Staubli VAL3: advance.pjx

--- advance.pjx ---
Parameters version=s7.2.1 stackSize=5000 millimeterUnit=true
Program file=findLastPathPos.pgx
Program file=language.pgx
Program file=loadPage.pgx
Program file=main.pgx
Program file=onEnterEvent.pgx
Program file=onExit.pgx
Program file=onF1Event.pgx
Program file=onF2Event.pgx
Program file=onF3Event.pgx
Program file=onF4Event.pgx
Program file=onF5Event.pgx
Program file=onF6Event.pgx
Program file=onF7Event.pgx
Program file=onF8Event.pgx
Program file=onStart.pgx
Program file=passwd.pgx
Program file=refresh.pgx
Program file=refreshDynamic.pgx
Program file=refreshExport.pgx
Program file=refreshImport.pgx
Program file=refreshStatic.pgx
Program file=settings.pgx
Data file=advance.dtx
Library alias=use path=Disk://kernel/userPage/userPage.pjx
Library alias=use2 path=Disk://kernel/userpage/userpage.pjx
Library alias=language path=Disk://kernel/language/language.pjx
Library alias=saveData path=Disk://saveData/saveData.pjx
Library alias=out path=Disk://instruction/inputOutput/OUT/OUT.pjx
Library alias=cycleStatus path=Disk://cycleStatus/cycleStatus.pjx
Library alias=tcp path=Disk://kernel/tool/tool.pjx
Library alias=page path=Disk://kernel/template/page/page.pjx
Type name=FrameItem path=Disk://kernel/template/FrameItem/FrameItem.pjx

--- advance.dtx ---
num nIndex
num nIndexExport
num nIndexImport
num nIndexPreset
num nKey
public num nPage
num nRefresh
num nTime = 1
num nView
num nViewExport
num nViewImport
string sEventExport
string sEventImport
string sExport
string sImport
public string sItems
string sMenu
string sMessage
string sMenu8[8]
bool bButton[8]
frame fFrame = {fatherId=world[0]}

--- main.pgx ---
public program main()
  local bool l_bSave
begin
  // INIT
  call onStart()
  // LOOP UNTIL nKey=255
  do
    call refresh()
    nKey=getKey()
    switch nKey
      case 271
        // GUN SELECTION
        call onF1Event(l_bSave)
      break
      case 272
        // LANGUAGE
        call onF2Event(l_bSave)
      break
      case 273
        //
        call onF3Event()
      break
      case 274
        //
        call onF4Event()
      break
      case 275
        //
        call onF5Event()
      break
      case 276
        // PLC
        call onF6Event(l_bSave)
      break
      case 277
        // PROFIILE
        call onF7Event(l_bSave)
      break
      case 278
        //
        call onF8Event()
      break
      case 270
        // NOTHING
        call onEnterEvent()
      break
    endSwitch
    //release the resource
    delay(0)
  until nKey==255
  // on Exit
  call onExit(l_bSave)
end

--- findLastPathPos.pgx ---
program findLastPathPos(string x_sPath (dimensions=1), num& x_nPos[] (dimensions=1))
  local num l_nPos[2]
  local string l_sPath
begin
  // get the trajType
  l_sPath=x_sPath
  x_nPos=0
  do
    l_nPos=find(l_sPath,"/")
    if l_nPos==-1
      l_nPos=find(l_sPath,"\")
    endIf
    if l_nPos!=-1
      x_nPos=x_nPos+l_nPos+1
      l_nPos[1]=l_nPos
      l_sPath=right(l_sPath,len(l_sPath)-l_nPos-1)
    endIf
  until l_nPos==-1
  // came back one
  x_nPos=x_nPos-l_nPos[1]-1
end

--- language.pgx ---
program language()
  local num l_nIndex
  local string l_sEvent
  local num i
  local string l_sMessage
begin
  //
  //  Select and change the language
  //
  call use:clear(0,13)
  call use:setView(false)
  // scan it
  libList(language:libPath(),sMessage)
  // clean
  for i=0 to size(sMessage)-1
    if find(sMessage[i],".")!=-1
      delete(sMessage[i])
      i=i-1
    endIf
  endFor
  call language:message(l_sMessage,50)
  call use:setSizeList(19,0,19,11)
  call use:listcreate(l_sMessage)
  // show it
  for i=0 to (size(sMessage)-1)
    l_sEvent=sMessage[i]
    call use:listadd(l_sEvent)
    if saveData:language==sMessage[i]
      l_nIndex=i
    endIf
  endFor
  // update the list
  use:nView=l_nIndex
  call use:listupdate(0)
  // scan for a button
  do
    i=get()
    call use:listevent(i,l_nIndex,l_sEvent)
  until i==270 or i==255
  if (i==270) and l_nIndex!=-1
    saveData:language=l_sEvent
    logMsg("[KERNEL] INTERFACE:Change language to "+l_sEvent)
    // set the language
    call language:setLanguage(language:libPath()+"/"+saveData:language)
  else
    call use:nullKey(i)
  endIf
end

--- loadPage.pgx ---
program loadPage(string x_sPage, string& x_sItems[])
// load the next page
  local num i
  local string l_sMessage
begin
  // look if the page libload is correct
  i=page:libLoad(x_sPage)
  delay(0)
  if i!=0
    logMsg("[KERNEL] INTERFACE:PAGE LIBLOAD "+x_sPage+" result "+toString("",i))
    call language:message(l_sMessage,-7)
    popUpMsg(l_sMessage+x_sPage+" ; "+toString("",i))
  else
    // copy all the field from x_sItems to the next page
    call use:stringCopy(x_sItems,page:sItems)
    call page:main()
  endIf
end

--- onEnterEvent.pgx ---
program onEnterEvent()
begin
  //
end

--- onExit.pgx ---
program onExit(bool x_bSave (dimensions=1))
  local num i
begin
  // save the saveData module
  if x_bSave
    if saveData:libSave()!=0
      delay(0.5)
      i=saveData:libSave()
      if i!=0
        popUpMsg("libsave saveData error: "+toString("",i))
        logMsg("[KERNEL] ADVANCE:Error saving saveData "+toString("",i))
      endIf
    endIf
  endIf
  //
  call use:nullKey(nKey)
end

--- onF1Event.pgx ---
program onF1Event(bool& x_bSave[])
  local string l_sParameter
  local string l_sItem
  local num l_nKey
  local num l_nIndex
  local string l_sPage
  local string l_sEvent
  local num i
begin
  // look if the bButton is enable
  if bButton[0]
    //
    // TOOL / FRAME SELECTION
    //
    call use:setSizeList(0,9,10,2)
    call use:listcreate("")
    // TOOL
    call language:message(l_sItem,124)
    call use:listadd(l_sItem)
    l_sItem="FRAME"
    call use:listadd(l_sItem)
    call use:listupdate(0)
    // get the key
    do
      l_nKey=get()
      call use:listevent(l_nKey,l_nIndex,l_sEvent)
    until l_nKey==270 or l_nKey==255
    // check the Enter key pressure
    if l_nKey==270
      switch l_nIndex
        case 0
          // Select the tool
          l_sPage="Disk://kernel/page/tool"
          call loadPage(l_sPage,l_sItem)
        break
        case 1
          // Select the Frame
          l_sPage="Disk://kernel/page/frame"
          call loadPage(l_sPage,l_sItem)
        break
      endSwitch
    endIf
    logMsg("[KERNEL] INTERFACE:PAGE Advance")
    x_bSave=true
  endIf
end

--- onF2Event.pgx ---
program onF2Event(bool& x_bSave[] (dimensions=1))
begin
  // look if the bButton is enable
  if bButton[1]
    //
    // CHANGE THE settings
    //
    setTextMode(1)
    call use:type(0,4,"F2 "+sMenu[1])
    setTextMode(0)
    call settings()
    use:bUseRefresh=true
    x_bSave=true
  endIf
end

--- onF3Event.pgx ---
program onF3Event()
  local string l_sMessage[2]
  local bool l_bImport
  local string l_sPath[2]
  local num l_nKey
  local bool l_bDone
  local num l_nOldValue[4]
  local num i
  local string l_sButton[2]
  local string l_sItem
  local string l_sType
begin
  //
  // look if the bButton is enable
  if bButton[2]
    if libList("USB0://",sImport)
      l_bImport=false
      //
      //  importing file
      //
      // get the path
      l_sPath="Disk://../usrapp/"
      //
      l_sPath[1]="USB0://"
      //
      title("< RESTORE / BACKUP >")
      cls()
      // copy the value
      l_nOldValue[2]=nIndexImport
      l_nOldValue[3]=nViewImport
      l_nOldValue=nIndex=0
      l_nOldValue[1]=nView
      //
      // IMPORT
      call use2:setSizeList(0,0,17,11)
      call use2:listcreate("USB")
      // paste the value
      nIndexImport=l_nOldValue[2]
      nViewImport=l_nOldValue[3]
      call refreshImport(false,l_sPath)
      // EXPORT
      call use:setSizeList(19,0,19,11)
      call use:listcreate("ROBOT")
      // paste the value
      nIndex=l_nOldValue=0
      nView=l_nOldValue[1]
      call refreshExport(true,l_sPath)
      l_sType="<<<<"
      call use:type(17,12,l_sType)
      //
      do
        call use:clear(0,13)
        call use:typeMenu(8,"COPY")
        l_nKey=get()
        switch l_nKey
          case 264
            l_bImport=true
            //refresh
            call refreshExport(false,l_sPath)
            call refreshImport(true,l_sPath)
            l_sType=">>>>"
            call use:type(17,12,l_sType)
          break
          case 268
            l_bImport=false
            //refresh
            //call refreshExport(true,l_sPath)
            call refreshImport(false,l_sPath)
            call refreshExport(true,l_sPath)
            l_sType="<<<<"
            call use:type(17,12,l_sType)
          break
        endSwitch
        // swich from import to export
        if l_bImport
          //
          // IMPORT
          //
          call use2:listevent(l_nKey,nIndexImport,sEventImport)
          nViewImport=use2:nView
          //
          if l_nKey>=259 and l_nKey<=278
            if l_nKey==278
              // look for already exist
              l_bDone=true
              for i=0 to size(sExport)-1
                if sExport[i]==sEventImport
                  call language:message(l_sMessage,11)
                  // get the yes_no button Key
                  call language:getYesNo(l_sButton)
                  // ask the question
                  call use:yes_no(l_sMessage+"#"+l_sPath+sEventImport,l_sButton,l_bDone)
                  i=size(sExport)-1
                endIf
              endFor
              //
              if l_bDone
                call language:message(l_sMessage,10)
                // show that will take several minute
                if find(sEventExport,"usrapp")!=-1
                  call language:message(l_sMessage[1],-9)
                  l_sMessage=l_sMessage+"#"+l_sMessage[1]
                endIf
                call use:timerDialog(l_sMessage+"#"+l_sPath+sEventImport,0)
                l_bDone=$copy(l_sPath[1]+sEventImport,l_sPath+sEventImport)
                if !l_bDone
                  call language:message(l_sMessage,-6)
                  call use:timerDialog(l_sMessage+"#"+l_sPath+sEventImport,2)
                endIf
              endIf
              // refresh backward
              cls()
              call refreshExport(false,l_sPath)
              call refreshImport(true,l_sPath)
              l_sType=">>>>"
              call use:type(17,12,l_sType)
            endIf
          endIf
          //
        else
          //
          //  EXPORT
          //
          call use:listevent(l_nKey,nIndex,sEventExport)
          nView=use:nView
          //
          if l_nKey>=259 and l_nKey<=278
            if l_nKey==278
              // look for already exist
              l_bDone=true
              for i=0 to size(sImport)-1
                if sImport[i]==sEventExport
                  call language:message(l_sMessage,11)
                  // get the yes_no button Key
                  call language:getYesNo(l_sButton)
                  // ask the question
                  call use:yes_no(l_sMessage+"#"+l_sPath+sEventExport,l_sButton,l_bDone)
                  i=size(sImport)-1
                endIf
              endFor
              if l_bDone
                call language:message(l_sMessage,10)
                // show that will take several minute
                if find(sEventExport,"usrapp")!=-1
                  call language:message(l_sMessage[1],-9)
                  l_sMessage=l_sMessage+"#"+l_sMessage[1]
                endIf
                // patch version 7
                if l_sPath=="Disk://../../"
                  l_sPath="Disk://../"
                endIf
                call use:timerDialog(l_sMessage+"#"+l_sPath[1]+sEventExport,0)
                l_bDone=$copy(l_sPath+sEventExport,l_sPath[1]+sEventExport)
                if !l_bDone
                  l_sMessage=l_sMessage+"#"+l_sPath[1]+sEventExport
                  call language:message(l_sMessage,-6)
                  call use:timerDialog(l_sMessage,2)
                endIf
                // patch version 7
                if l_sPath=="Disk://../"
                  l_sPath="Disk://../../"
                endIf
              endIf
              // refresh backward
              cls()
              call refreshImport(false,l_sPath)
              call refreshExport(true,l_sPath)
              l_sType="<<<<"
              call use:type(17,12,l_sType)
            endIf
            //
          endIf
        endIf
        // NAVIGATION
        if l_nKey==270
          if l_bImport
            // IMPORT BOX
            if sEventImport==".."
              call findLastPathPos(l_sPath[1],i)
              l_sPath[1]=left(l_sPath[1],i)
            else
              l_sPath[1]=l_sPath[1]+sEventImport+"/"
            endIf
            // refresh IMPORT
            nIndexImport=nViewImport=use2:nView=0
            call refreshImport(true,l_sPath)
          else
            // EXPORT BOX
            if sEventExport==".."
              call findLastPathPos(l_sPath,i)
              l_sPath=left(l_sPath,i)
              // patch version 7
              if l_sPath=="Disk://../"
                l_sPath="Disk://../../"
              endIf
            else
              if l_sPath=="Disk://../../"
                l_sPath="Disk://../"
              endIf
              l_sPath=l_sPath+sEventExport+"/"
            endIf
            // refresh EXPORT
            nIndex=nView=use:nView=0
            call refreshExport(true,l_sPath)
          endIf
        endIf
        //
      until l_nKey==255
      //
      call refreshStatic()
      //
    else
      // NO USB in the controller
      call language:message(l_sMessage,-10)
      popUpMsg(l_sMessage)
    endIf
  endIf
end

--- onF4Event.pgx ---
program onF4Event()
begin
  // look if the bButton is enable
  if bButton[3]
    // F4 Button
  endIf
end

--- onF5Event.pgx ---
program onF5Event()
  local string l_sItem
begin
  // look if the bButton is enable
  if bButton[4]
    //
    logMsg("[KERNEL] INTERFACE:PAGE Advance")
  endIf
end

--- onF6Event.pgx ---
program onF6Event(bool& x_bSave[] (dimensions=1))
begin
  // look if the bButton is enable
  if bButton[5] and saveData:mode>1
    //
    // CHANGE PLC STATUS
    //
    if saveData:bPlc
      cycleStatus:nInterfaceToSV=11
    else
      cycleStatus:nInterfaceToSV=10
    endIf
    wait(cycleStatus:nInterfaceToSV==-1)
    logMsg("[KERNEL] INTERFACE:Change PLC STATUS")
    x_bSave=true
  endIf
end

--- onF7Event.pgx ---
program onF7Event(bool& x_bSave[] (dimensions=1))
begin
  // look if the bButton is enable
  if bButton[6]
    //
    // CHANGE THE PROFILE
    //
    call passwd(x_bSave)
  endIf
end

--- onF8Event.pgx ---
program onF8Event()
  local string l_sItem
begin
  // look if the bButton is enable
  if bButton[7]
    //
    call loadPage("Disk://trajectory/TRACK/page_viewTrack",l_sItem)
    logMsg("[KERNEL] INTERFACE:PAGE Advance")
  endIf
end

--- onStart.pgx ---
program onStart()
  local num l_nSize
  local frame l_fNewWorld
begin
  // load the default gun
  if !cycleStatus:bCycle
    call tcp:getSize(l_nSize)
    if saveData:nIndexTool>=l_nSize
      // BAD GUN INDEX load default ZERO
      saveData:nIndexTool=0
    endIf
    // get the tool
    call tcp:getTool(saveData:tTool,saveData:nIndexTool)
    fFrame.trsf=saveData:fFrameItem[saveData:nFrameActive].fFrame.trsf
    $jogContext(saveData:tTool,fFrame,0)
  endIf
  //
  // logMsg
  logMsg("[KERNEL] INTERFACE:PAGE Advance")
  //
  use:bUseRefresh=true
end

--- passwd.pgx ---
program passwd(bool& x_bSave[] (dimensions=1))
  local string sText
  local string sTempMessage
  local num i
  local string message
begin
  //
  // clean the screen
  //
  cls()
  call language:message(message,204)
  call use:timerDialog(message,0)
  call use:type(2,8,">")
  call use:read(3,8,sText,15,true)
  //
  // there are 3 difference kind of access
  // mode 0   ->operator
  // mode 1   ->programmer
  // mode 2   ->integrator
  // mode 3   ->toneage (Administrator)
  //
  saveData:mode=0
  for i=0 to (size(saveData:passwd)-1)
    if sText==saveData:passwd[i]
      saveData:mode=i+1
      call use:type(20,8,"...OK...")
      logMsg("[KERNEL] INTERFACE:Set password to: "+sText)
    endIf
  endFor
  if saveData:mode==0
    logMsg("[KERNEL] INTERFACE:Set password to: Operator")
  endIf
  //
  // It's possible to change the password
  //
  if saveData:mode>0 and saveData:mode<3
    call language:message(message,205)
    call use:type(0,10,message)
    call language:message(message,206)
    call use:typeMenu(5,message)
    call use:typeMenu(8,"OK")
    nKey=get()
    if nKey==275
      cls()
      call language:message(message,207)
      call use:timerDialog(message,0)
      call use:type(2,8,">")
      sText=""
      call use:read(3,8,sText,15,true)
      call language:message(message,208)
      call use:timerDialog(message,0)
      sTempMessage=""
      call use:read(3,8,sTempMessage,15,true)
      //
      // look if the passwd already exist
      //
      if sText==sTempMessage and sText!=""
        if saveData:passwd[0]!=sText and saveData:passwd[1]!=sText
          saveData:passwd[saveData:mode-1]=sText
        else
          call language:message(message,-2)
          popUpMsg(message)
        endIf
      else
        call language:message(message,209)
        popUpMsg(message)
      endIf
    endIf
  endIf
  //
  //  Show your mode to access and set the Userpage
  //
  switch saveData:mode
    case 0
      call language:message(sText,210)
    break
    case 1
      call language:message(sText,211)
    break
    case 2,3
      call language:message(sText,212)
    break
  endSwitch
  if saveData:mode<2
    userPage(true)
  else
    userPage(false)
  endIf
  call language:message(message,213)
  popUpMsg(message+sText)
  // SAVE THE SETTING
  x_bSave=true
  //
  nKey=255
end

--- refresh.pgx ---
program refresh()
// // page refresh
begin
  // refresh the static message
  if (nKey>=270 and nKey<=278) or use:bUseRefresh
    call refreshStatic()
    call refreshDynamic()
  else
    // refresh the Dynamic message
    if abs(clock()-nRefresh)>nTime
      call refreshDynamic()
    endIf
  endIf
end

--- refreshDynamic.pgx ---
program refreshDynamic()
begin
  // DO NOT CHANGE
  nRefresh=clock()
  use:bUseRefresh=false
  //
  // ADD HERE
  //
end

--- refreshExport.pgx ---
program refreshExport(bool x_bShowLine (dimensions=1), string x_sPath (dimensions=1))
  local num l_nLocal
  local string l_sEmpty
  local string l_sItem
begin
  call use:setSizeList(19,0,19,11)
  call use:listcreate("ROBOT")
  call use:stringCopy(l_sEmpty,sExport)
  call use:listempty()
  //
  // build the list
  if libList(x_sPath,sExport)
    // build and refresh
    if x_sPath!="Disk://../"
      l_sItem=".."
      call use:listadd(l_sItem)
    endIf
    call use:listadd(sExport)
    use:nView=nView
    call use:listredraw(nIndex-nView)
    if !x_bShowLine
      call use:listcursor(nView,false)
    endIf
  endIf
end

--- refreshImport.pgx ---
program refreshImport(bool x_bShowLine (dimensions=1), string& x_sPath[] (dimensions=1))
  local num l_nLocal
  local string l_sEmpty
  local string l_sItem
begin
  //
  call use2:setSizeList(0,0,17,11)
  call use2:listcreate("USB")
  call use:stringCopy(l_sEmpty,sImport)
  call use2:listempty()
  //
  // build the list
  if libList(x_sPath[1],sImport)
    // build and refresh
    if x_sPath[1]!="USB0://"
      l_sItem=".."
      call use2:listadd(l_sItem)
    endIf
    call use2:listadd(sImport)
    use2:nView=nViewImport
    call use2:listredraw(nIndexImport-nViewImport)
    if !x_bShowLine
      call use2:listcursor(nViewImport,false)
    endIf
  endIf
end

--- refreshStatic.pgx ---
program refreshStatic()
  local string l_sString
  local string l_sPreset[3]
  local string l_sMessage
  local bool l_bOutMode[6]
  local string l_sName
begin
  cls()
  //
  // set the view of the page..
  //
  // SET THE PAGE NUMBER
  use:nPage=140
  // USE <>PROFILE for <>PAGE
  use:nPage=use:nPage+abs(limit(saveData:mode,0,2)-2)
  //
  if cycleStatus:bCycle
    use:nPage=use:nPage+3
  endIf
  if saveData:language!="japanese"
    // SET THE VIEW OF THE PAGE
    call language:page(l_sMessage,use:nPage)
    // define the menu
    call use:stringToArray(l_sMessage,sMenu)
  else
    // japanese use the array for the menu
    call language:page(sMenu8,use:nPage)
    call use:stringCopy(sMenu8,sMenu)
  endIf
  //
  //
  // TOOL
  //
  call language:message(l_sMessage,124)
  call tcp:getName(l_sName,saveData:nIndexTool)
  call use:type(18,2,"┌-> "+l_sMessage+":"+toString("",saveData:nIndexTool)+" "+l_sName)
  call language:message(l_sMessage,124)
  l_sName=saveData:fFrameItem[saveData:nFrameActive].sName
  call use:type(18,3,"--> Frame:"+toString("",saveData:nFrameActive)+" "+l_sName)
  //
  //  PLC
  //
  if saveData:bPlc
    call use:type(18,8,"--> ON ")
  else
    call use:type(18,8,"--> OFF")
  endIf
  // Profile
  //
  // switch case mode
  //
  call language:message(l_sString,limit(saveData:mode,0,2))
  call use:type(18,9,"-->"+l_sString)
  //
  if !cycleStatus:bTrackEnable
    sMenu[7]=""
  endIf
  //
  // define the bButton and Menu
  call use:setMenu(sMenu,false,3)
  call use:getMenu(sMenu,bButton)
end

--- settings.pgx ---
program settings()
  local string l_sEvent
  local num l_nIndex
  local num i
  local string l_sMessage
  local string l_sItem
  local string l_sEmpty
begin
  // set the items
  call use:clear(0,13)
  // show the items
  do
    // build the list
    call use:setSizeList(16,3,22,8)
    call use:listcreate("")
    // language
    call language:message(l_sMessage,50)
    l_sMessage=l_sMessage+"> "+saveData:language
    call use:listadd(l_sMessage)
    // rounding
//    call language:message(l_sMessage,51)
//    l_sMessage=l_sMessage+"> "+toString("",saveData:nRound)+"%"
//    call use:listadd(l_sMessage)
//    // timeOut
//    call language:message(l_sMessage,52)
//    if saveData:nTimeOut>0
//      l_sItem="[x]"+l_sMessage+"> "+toString("",saveData:nTimeOut)+" sec."
//    else
//      l_sItem="[ ]"+l_sMessage+">     "
//    endIf
//    call use:listadd(l_sItem)
//    // multiSession
//    call use:showBoolStatus(saveData:bMultiSession,l_sItem)
//    call language:message(l_sMessage,53)
//    l_sMessage=l_sItem+l_sMessage
//    call use:listadd(l_sMessage)
//    // Reload the last saved process List
//    call language:message(l_sMessage,55)
//    call use:showBoolStatus(saveData:bReloadList,l_sItem)
//    l_sMessage=l_sItem+l_sMessage
//    call use:listadd(l_sMessage)
//    // set the timer Dialog joint/Frame status
//    call language:message(l_sMessage,54)
//    if saveData:nTimeDialog>0
//      l_sItem="[x]"+l_sMessage+"> "+toString("",saveData:nTimeDialog)+" sec."
//    else
//      l_sItem="[ ]"+l_sMessage+">     "
//    endIf
//    call use:listadd(l_sItem)
//    // add the stop on power Off
//    call language:message(l_sMessage,56)
//    call use:showBoolStatus(saveData:bStopToPowerOff,l_sItem)
//    l_sMessage=l_sItem+l_sMessage
//    call use:listadd(l_sMessage)
//    // show nested data
//    call use:showBoolStatus(saveData:bShowItem,l_sItem)
//    call language:message(l_sMessage,57)
//    l_sMessage=l_sItem+l_sMessage
//    call use:listadd(l_sMessage)
    // refresh the list
    call use:listupdate(0)
    nKey=get()
    call use:listevent(nKey,l_nIndex,l_sEvent)
    switch nKey
      // ENTER KEY
      case 270
        call use:findPos(l_sEvent,">",i)
        // list cursor to false
        call use:listcursor(l_nIndex,false)
        // switch it
        switch l_nIndex
          case 0
            // change the language
            call language()
            return
          break
          case 1
            // change the rounding correction
            l_sEmpty=""
            call use:changeValue(saveData:nRound,0,100,use:nTopX+i+2+1,use:nTopY+l_nIndex+1,l_sEmpty)
          break
          case 2
            // change the timeout event
            l_sEmpty=""
            call use:changeValue(saveData:nTimeOut,0,999,use:nTopX+i+2+1,use:nTopY+l_nIndex+1,l_sEmpty)
          break
          case 3
            // change the multisession
            saveData:bMultiSession=!saveData:bMultiSession
          break
          case 4
            // change the multi processList
            saveData:bReloadList=!saveData:bReloadList
          break
          case 5
            // change the timeout event
            l_sEmpty=""
            call use:changeValue(saveData:nTimeDialog,0,999,use:nTopX+i+2+1,use:nTopY+l_nIndex+1,l_sEmpty)
          break
          case 6
            // STOP on Lost Power OFF
            saveData:bStopToPowerOff=!saveData:bStopToPowerOff
          break
          case 7
            // show nested element
            saveData:bShowItem=!saveData:bShowItem
          break
        endSwitch
      break
      // SPACE KEY
      case 32
        switch l_nIndex
          case 2
            // time Out
            saveData:nTimeOut=-saveData:nTimeOut
          break
          case 3
            // change the multisession
            saveData:bMultiSession=!saveData:bMultiSession
          break
          case 4
            // change the multi processList
            saveData:bReloadList=!saveData:bReloadList
          break
          case 5
            // time Out
            saveData:nTimeDialog=-saveData:nTimeDialog
          break
          case 6
            // STOP on Lost Power OFF
            saveData:bStopToPowerOff=!saveData:bStopToPowerOff
          break
          case 7
            // show nested element
            saveData:bShowItem=!saveData:bShowItem
          break
        endSwitch
      break
    endSwitch
  until nKey==255
  // release
  call use:nullKey(nKey)
end
